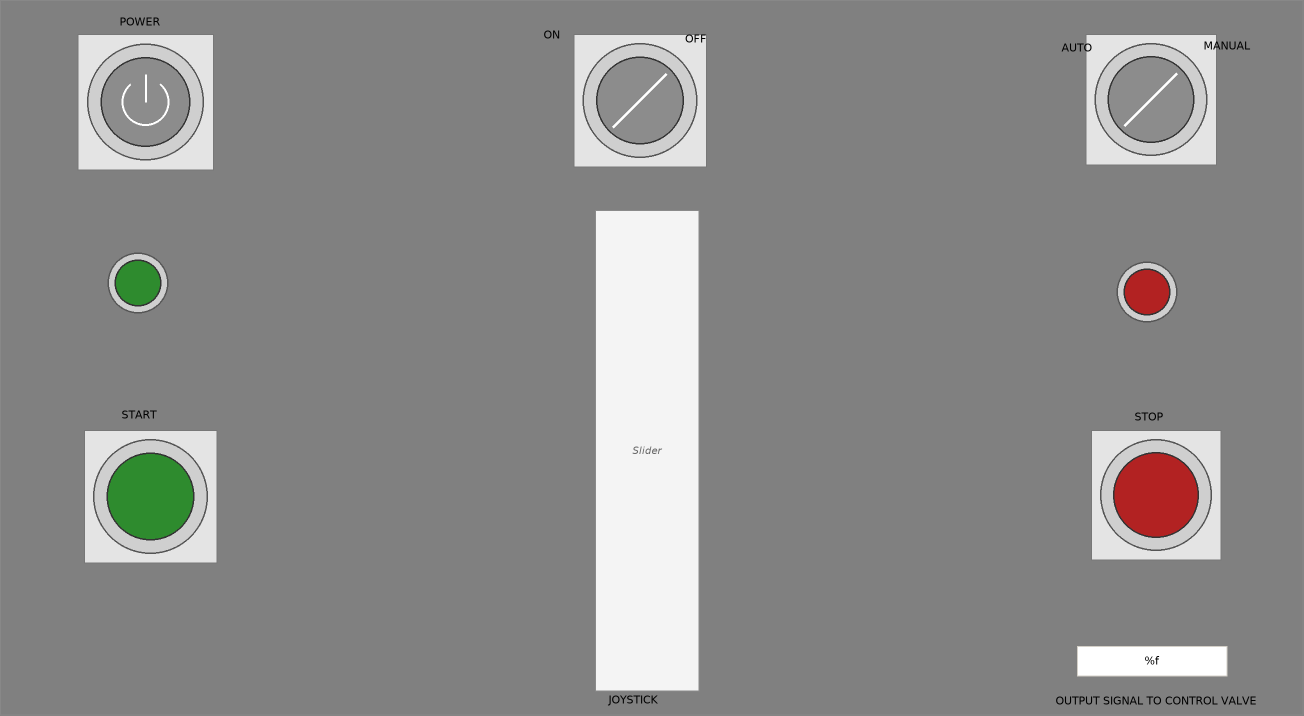
VISUALIZATION HMI  // 1304x716
    PowerSwitch (75,34 141x136), variable: HMIinput.bHMIPowerSwitch, behaviour: TOGGLE, style: Switch-PowerSwitch-Gray
    PushSwitch (74,430 153x133), variable: HMIinput.bHMIStartSwitch, behaviour: TOGGLE, style: Switch-PushSwitch-Green
    PushSwitch (1085,430 142x130), variable: HMIinput.bHMIStopSwitch, behaviour: TOGGLE, style: Switch-PushSwitch-Red
    RotarySwitch (566,34 148x133), variable: HMIinput.bHMIOnOffSwitch, behaviour: TOGGLE, style: Switch-RotarySwitch-Gray
    RotarySwitch (1085,34 132x131), variable: HMIinput.bHMIModeSwitch, behaviour: TOGGLE, style: Switch-RotarySwitch-Gray
    Slider (595,210 104x481), variable: MAIN.fPodMeas, scale -1..1
    Label (1002,33 150x30), "AUTO"
    Label (1074,402 150x30), "STOP"
    Label (1152,31 150x30), "MANUAL"
    Label (477,20 150x30), "ON"
    Label (621,24 150x30), "OFF"
    Label (64,400 150x30), "START"
    Label (65,7 150x30), "POWER"
    Lamp1 (103,248 70x70), variable: HMIoutput.bHMIGreenLED, style: Lamp-Lamp1-Green
    Lamp1 (1112,257 70x70), variable: HMIoutput.bHMIRedLED, style: Lamp-Lamp1-Red
    Textfield (1077,646 150x30), "%f", text variable: HMIoutput.fHMIControlValveSignal
    Label (1008,686 296x30), "OUTPUT SIGNAL TO CONTROL VALVE"
    Label (558,685 150x30), "JOYSTICK"
END_VISUALIZATION

(* stored: Version 1.1.0.1, ProductVersion 3.1.4024.10
   Visu HMI: Id {13dbd610-74c1-4a63-80d9-d312b3110d4a} *)
